// TIA Portal project "washing machine" (V16)

(* hardware
DEVICE "S7-1200 station_1"  S7-1200 Station
   slot 0: "Rack_0"  S7-1200 Rack  Rack  V1.0
   slot 1: "PLC_1"  CPU 1212C AC/DC/Rly  6ES7 212-1BE40-0XB0  V4.0
*)

// ===== PLC "PLC_1"  CPU 1212C AC/DC/Rly =====

VAR_GLOBAL   // PLC tag table "Default tag table"
   "stop" AT %I0.0 : Bool;
   "start" AT %I0.1 : Bool;
   "Forward" AT %Q0.0 : Bool;
   "reverse" AT %Q0.2 : Bool;
   "loop marker" AT %M0.0 : Bool;
   "delay1" AT %M0.1 : Bool;
   "delay2" AT %M0.2 : Bool;
END_VAR

// folder: System blocks/Program resources

DATA_BLOCK "T1"   // DB1
{ S7_Optimized_Access := 'TRUE' }
AUTHOR : Simatic
FAMILY : IEC
NAME : IEC_TMR
VERSION : 1.0
// stored: InstanceOfName IEC_TIMER
"IEC_TIMER"
BEGIN
END_DATA_BLOCK

DATA_BLOCK "DT2"   // DB2
{ S7_Optimized_Access := 'TRUE' }
AUTHOR : Simatic
FAMILY : IEC
NAME : IEC_TMR
VERSION : 1.0
// stored: InstanceOfName IEC_TIMER
"IEC_TIMER"
BEGIN
END_DATA_BLOCK

DATA_BLOCK "T2"   // DB3
{ S7_Optimized_Access := 'TRUE' }
AUTHOR : Simatic
FAMILY : IEC
NAME : IEC_TMR
VERSION : 1.0
// stored: InstanceOfName IEC_TIMER
"IEC_TIMER"
BEGIN
END_DATA_BLOCK

DATA_BLOCK "DT4"   // DB4
{ S7_Optimized_Access := 'TRUE' }
AUTHOR : Simatic
FAMILY : IEC
NAME : IEC_TMR
VERSION : 1.0
// stored: InstanceOfName IEC_TIMER
"IEC_TIMER"
BEGIN
END_DATA_BLOCK

// folder: (top level)

ORGANIZATION_BLOCK "Main"   // OB1, LAD, ProgramCycle
TITLE = "Main Program Sweep (Cycle)"
{ S7_Optimized_Access := 'TRUE' }
VERSION : 0.1
   VAR_INPUT
      Initial_Call : Bool;   // Initial call of this OB
      Remanence : Bool;   // =True, if remanent data are available
   END_VAR
BEGIN

REGION Network 1
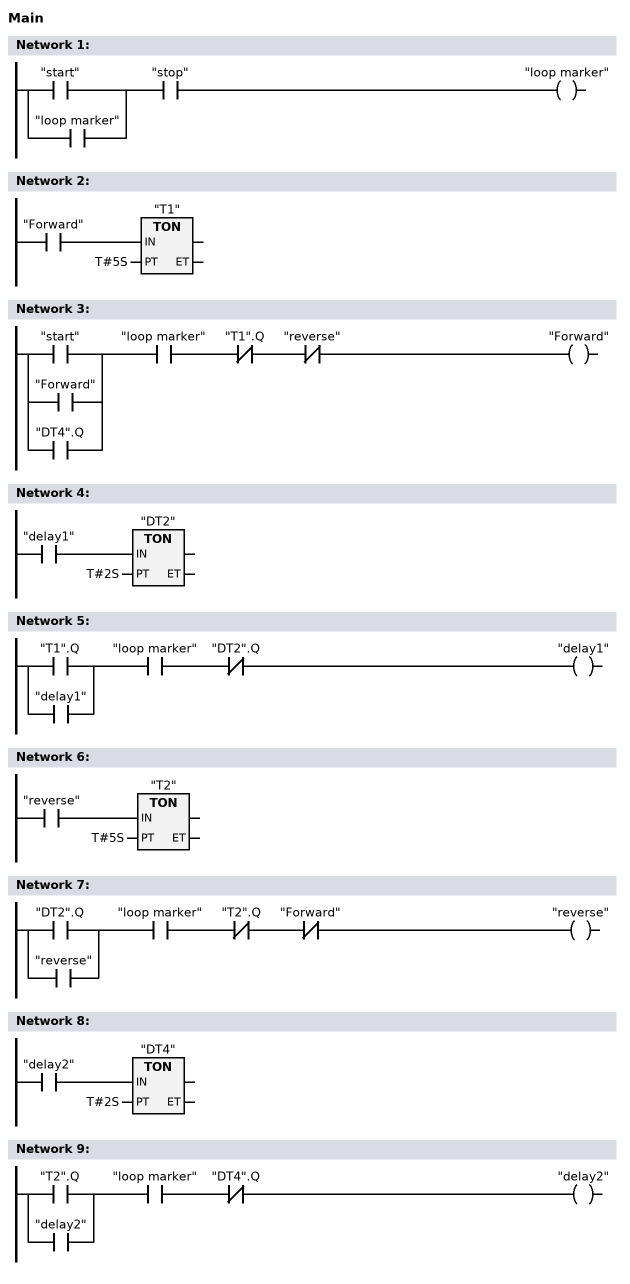
   RUNG wire#powerrail
      Contact( "start" )
      wire#w1
      Contact( "stop" )
      Coil( "loop marker" )
   END_RUNG
   RUNG wire#powerrail
      Contact( "loop marker" )
   END_RUNG wire#w1
   // the same network as SCL:
   "loop marker" := ("start" OR "loop marker") AND "stop";
END_REGION

REGION Network 2
   "T1".TON(IN := "Forward", PT := T#5S);
END_REGION

REGION Network 3
   RUNG wire#powerrail
      Contact( "start" )
      wire#w1
      Contact( "loop marker" )
      I_Contact( "T1".Q )
      I_Contact( "reverse" )
      Coil( "Forward" )
   END_RUNG
   RUNG wire#powerrail
      Contact( "Forward" )
   END_RUNG wire#w1
   RUNG wire#powerrail
      Contact( "DT4".Q )
   END_RUNG wire#w1
   // the same network as SCL:
   "Forward" := ("start" OR "Forward" OR "DT4".Q) AND "loop marker" AND NOT "T1".Q AND NOT "reverse";
END_REGION

REGION Network 4
   "DT2".TON(IN := "delay1", PT := T#2S);
END_REGION

REGION Network 5
   RUNG wire#powerrail
      Contact( "T1".Q )
      wire#w1
      Contact( "loop marker" )
      I_Contact( "DT2".Q )
      Coil( "delay1" )
   END_RUNG
   RUNG wire#powerrail
      Contact( "delay1" )
   END_RUNG wire#w1
   // the same network as SCL:
   "delay1" := ("T1".Q OR "delay1") AND "loop marker" AND NOT "DT2".Q;
END_REGION

REGION Network 6
   "T2".TON(IN := "reverse", PT := T#5S);
END_REGION

REGION Network 7
   RUNG wire#powerrail
      Contact( "DT2".Q )
      wire#w1
      Contact( "loop marker" )
      I_Contact( "T2".Q )
      I_Contact( "Forward" )
      Coil( "reverse" )
   END_RUNG
   RUNG wire#powerrail
      Contact( "reverse" )
   END_RUNG wire#w1
   // the same network as SCL:
   "reverse" := ("DT2".Q OR "reverse") AND "loop marker" AND NOT "T2".Q AND NOT "Forward";
END_REGION

REGION Network 8
   "DT4".TON(IN := "delay2", PT := T#2S);
END_REGION

REGION Network 9
   RUNG wire#powerrail
      Contact( "T2".Q )
      wire#w1
      Contact( "loop marker" )
      I_Contact( "DT4".Q )
      Coil( "delay2" )
   END_RUNG
   RUNG wire#powerrail
      Contact( "delay2" )
   END_RUNG wire#w1
   // the same network as SCL:
   "delay2" := ("T2".Q OR "delay2") AND "loop marker" AND NOT "DT4".Q;
END_REGION
END_ORGANIZATION_BLOCK